ABB RobotStudio station: dispencing_hg.rsstn

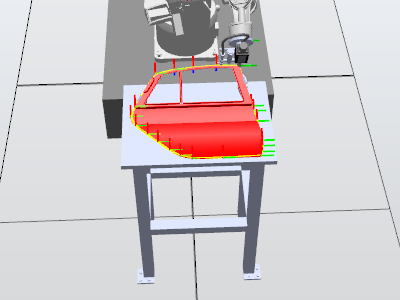
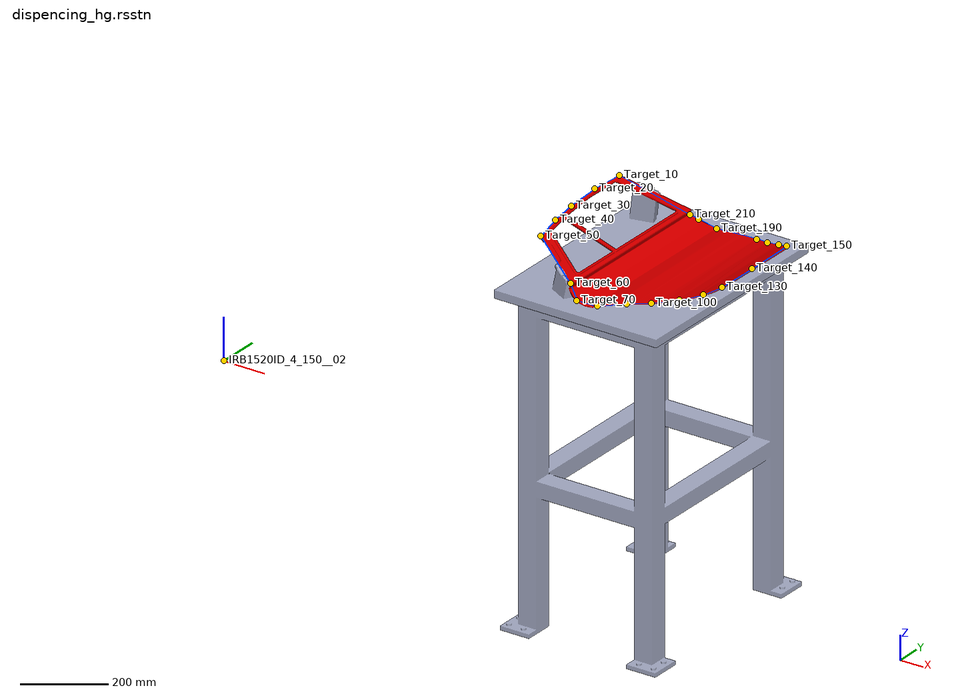
[picture v1: parts stored in the station drawn from their meshes, with robot base, taught points and paths (robot models come from the ABB library and are not in the file)]
Station Station (saved by RobotStudio 22.3.10141.1)
Controller Controller12, task T_ROB1: task frame (RAPID world) sits at (0, 0, 300) mm in the station
Controller Controller12
  mechanical unit ROB_1: IRB1520ID_4_150__02, 6 joints, base frame (0, 0, 0) mm
Layout (positions relative to the parent item):
  - IRB1520ID_4_150__02 [mechanism, from Robots\IRB1520ID_4_150_G_02.rslib] at (0, 0, 300) mm; joint values [0.2414, -0.1124, 0.5555, -1.1561, 0.2282, 1.2688] (rad or m)
  - Concrete 2 [part, from Libraries\Concrete 2.rslib] at (-450, -450, 0) mm
  - Dispencer [mechanism, from Dispencing\Dispencer.rslib] at (981.81, 199.08, 1109.95) mm, rotated rx 180 ry 60 rz 180 deg
  - table with door_2 [part] at (1539.59, 277.82, 378.56) mm, rotated rx 90 ry 0 rz -90 deg, size 600 x 960.7 x 450 mm
Attachment: Dispencer is attached to IRB1520ID_4_150__02 / Link6
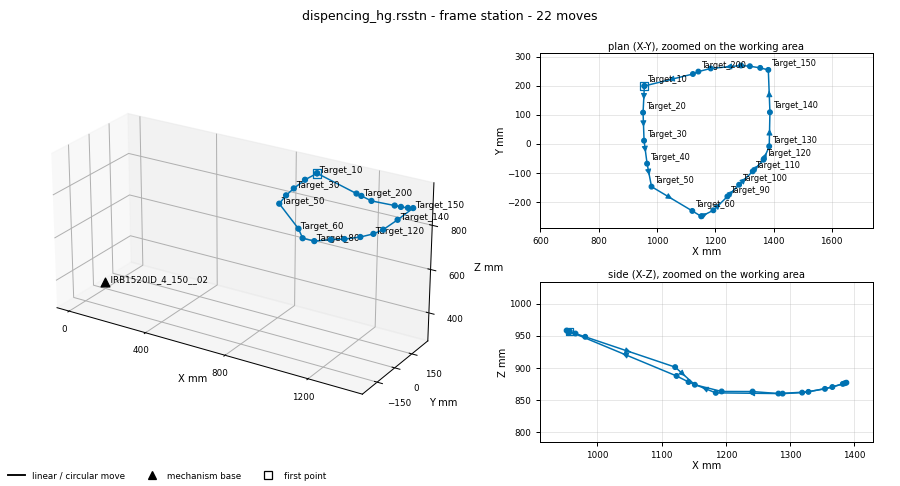
[picture p0: tool path of dispencing_hg.rsstn in frame station, 22 of 22 moves have a stored position in this frame; points joined in program order, loops and branches not executed]
Targets, tools, work objects and paths stored in the station, written as RAPID:
! task T_ROB1
MODULE CalibData
  PERS tooldata Dispencer:=[TRUE,[[145,-0.097,55],[0.707106781,0,0.707106781,0]],[1,[0,0,1],[1,0,0,0],0,0,0]];
ENDMODULE

! task T_ROB1
MODULE Module1
  CONST robtarget Target_10:=[[956.72339267,198.641198693,656.952986542],[0.258819024,0.000000009,-0.965925832,-0.000000029],[0,-1,0,0],[9E+09,9E+09,9E+09,9E+09,9E+09,9E+09]];
  CONST robtarget Target_20:=[[952.209475821,107.568800352,658.474636071],[0.258819021,0.000000009,-0.965925833,-0.000000033],[0,-1,0,0],[9E+09,9E+09,9E+09,9E+09,9E+09,9E+09]];
  CONST robtarget Target_30:=[[955.606400573,11.138031217,654.480276267],[0.258819031,0.000000009,-0.96592583,-0.000000034],[0,-1,0,0],[9E+09,9E+09,9E+09,9E+09,9E+09,9E+09]];
  CONST robtarget Target_40:=[[966.035312798,-67.831824904,653.814045381],[0.258819016,0.00000001,-0.965925834,-0.000000038],[-1,0,-1,0],[9E+09,9E+09,9E+09,9E+09,9E+09,9E+09]];
  CONST robtarget Target_50:=[[981.203616228,-146.67710529,648.700895808],[0.258819027,0.000000018,-0.965925831,-0.000000041],[-1,0,-1,0],[9E+09,9E+09,9E+09,9E+09,9E+09,9E+09]];
  CONST robtarget Target_60:=[[1121.216065138,-230.071220429,601.503386789],[0.258819025,0.000000043,-0.965925832,0.000000009],[-1,0,-1,0],[9E+09,9E+09,9E+09,9E+09,9E+09,9E+09]];
  CONST robtarget Target_70:=[[1151.783963237,-248.650796847,574.07892812],[0.258819022,0.000000018,-0.965925832,-0.00000008],[-1,0,-2,0],[9E+09,9E+09,9E+09,9E+09,9E+09,9E+09]];
  CONST robtarget Target_80:=[[1193.534985813,-227.921114684,563.642086785],[0.258819028,0.000000051,-0.965925831,0.000000038],[-1,1,-2,0],[9E+09,9E+09,9E+09,9E+09,9E+09,9E+09]];
  CONST robtarget Target_90:=[[1241.718073137,-180.459313001,563.500245858],[0.258819018,0.000000052,-0.965925834,0.000000017],[-1,0,-1,0],[9E+09,9E+09,9E+09,9E+09,9E+09,9E+09]];
  CONST robtarget Target_100:=[[1281.968020317,-140.115392307,560.348513441],[0.258819024,0.000000037,-0.965925832,-0.000000056],[-1,0,-1,0],[9E+09,9E+09,9E+09,9E+09,9E+09,9E+09]];
  CONST robtarget Target_110:=[[1328.622005559,-94.172884767,562.987416183],[0.258819014,0.000000036,-0.965925835,-0.000000056],[-1,0,-1,0],[9E+09,9E+09,9E+09,9E+09,9E+09,9E+09]];
  CONST robtarget Target_120:=[[1365.895055422,-54.093919947,570.51630961],[0.258819017,0.000000036,-0.965925834,-0.000000056],[-1,0,-1,0],[9E+09,9E+09,9E+09,9E+09,9E+09,9E+09]];
  CONST robtarget Target_130:=[[1385.27407376,-8.147577694,576.456220903],[0.258819015,0.000000036,-0.965925834,-0.000000056],[-1,0,-1,0],[9E+09,9E+09,9E+09,9E+09,9E+09,9E+09]];
  CONST robtarget Target_140:=[[1387.724068422,108.745605412,577.31184482],[0.258819012,0.000000038,-0.965925835,-0.000000058],[0,-1,0,0],[9E+09,9E+09,9E+09,9E+09,9E+09,9E+09]];
  CONST robtarget Target_150:=[[1382.166055675,254.129114737,575.40550814],[0.258819012,0.000000026,-0.965925835,-0.000000094],[0,-1,0,0],[9E+09,9E+09,9E+09,9E+09,9E+09,9E+09]];
  CONST robtarget Target_160:=[[1354.375981469,261.029520452,567.656223942],[0.258819023,0.000000025,-0.965925832,-0.000000105],[0,-1,0,0],[9E+09,9E+09,9E+09,9E+09,9E+09,9E+09]];
  CONST robtarget Target_170:=[[1318.858052657,266.752991236,561.823005064],[0.258819024,0.000000035,-0.965925832,-0.000000071],[0,-1,0,0],[9E+09,9E+09,9E+09,9E+09,9E+09,9E+09]];
  CONST robtarget Target_180:=[[1288.458007728,269.13699981,560.274801471],[0.258819022,0.000000034,-0.965925833,-0.000000068],[0,-1,0,0],[9E+09,9E+09,9E+09,9E+09,9E+09,9E+09]];
  CONST robtarget Target_190:=[[1184.389006392,259.073213384,561.468503207],[0.258819023,0.000000033,-0.965925832,-0.00000008],[0,-2,1,0],[9E+09,9E+09,9E+09,9E+09,9E+09,9E+09]];
  CONST robtarget Target_200:=[[1142.038949296,248.326203254,578.346383925],[0.258819027,0.000000023,-0.965925831,-0.000000109],[0,-1,1,0],[9E+09,9E+09,9E+09,9E+09,9E+09,9E+09]];
  CONST robtarget Target_210:=[[1123.353016328,240.045695555,587.742097013],[0.258819022,0.00000003,-0.965925833,-0.000000078],[0,-1,1,0],[9E+09,9E+09,9E+09,9E+09,9E+09,9E+09]];
  CONST robtarget Target_220:=[[956.939514886,198.980511555,656.880202244],[0.258819032,0.00000003,-0.96592583,-0.000000086],[0,-1,0,0],[9E+09,9E+09,9E+09,9E+09,9E+09,9E+09]];
  PROC Path_10()
    MoveL Target_10,v1000,z100,Dispencer\WObj:=wobj0;
    MoveL Target_20,v1000,z100,Dispencer\WObj:=wobj0;
    MoveL Target_30,v1000,z100,Dispencer\WObj:=wobj0;
    MoveL Target_40,v1000,z100,Dispencer\WObj:=wobj0;
    MoveL Target_50,v1000,z100,Dispencer\WObj:=wobj0;
    MoveL Target_60,v1000,z100,Dispencer\WObj:=wobj0;
    MoveL Target_70,v1000,z100,Dispencer\WObj:=wobj0;
    MoveL Target_80,v1000,z100,Dispencer\WObj:=wobj0;
    MoveL Target_90,v1000,z100,Dispencer\WObj:=wobj0;
    MoveL Target_100,v1000,z100,Dispencer\WObj:=wobj0;
    MoveL Target_110,v1000,z100,Dispencer\WObj:=wobj0;
    MoveL Target_120,v1000,z100,Dispencer\WObj:=wobj0;
    MoveL Target_130,v1000,z100,Dispencer\WObj:=wobj0;
    MoveL Target_140,v1000,z100,Dispencer\WObj:=wobj0;
    MoveL Target_150,v1000,z100,Dispencer\WObj:=wobj0;
    MoveL Target_160,v1000,z100,Dispencer\WObj:=wobj0;
    MoveL Target_170,v1000,z100,Dispencer\WObj:=wobj0;
    MoveL Target_180,v1000,z100,Dispencer\WObj:=wobj0;
    MoveL Target_190,v1000,z100,Dispencer\WObj:=wobj0;
    MoveL Target_200,v1000,z100,Dispencer\WObj:=wobj0;
    MoveL Target_210,v1000,z100,Dispencer\WObj:=wobj0;
    MoveL Target_220,v1000,z100,Dispencer\WObj:=wobj0;
  ENDPROC
ENDMODULE

